{attribute 'qualified_only'}
VAR_GLOBAL
		EtherCAT_Master_EKxxxx : EtherCAT_Master_EKxxxx_E740B17E;
END_VAR

(* stored: Version 1.2.0.0, ProductVersion 3.1.4024.9
   GVL GVL_iXlinker: Id {da893593-3b03-4825-8701-5760f119293a} *)
